PROGRAM MAIN
VAR
	a: int ;
END_VAR

Prg_Test();

a:= a+1;

END_PROGRAM

(* stored: Version 1.1.0.1
   POU MAIN: Id {85f428d9-07aa-4c8b-ba82-a8bb0d982cb1}, SpecialFunc None *)
